{attribute 'reflection'} 
FUNCTION_BLOCK FB_Component IMPLEMENTS I_Component
VAR_INPUT
	fbInfo:						FB_Info(sInstancePath, eState);
	fbEvent:					FB_Event(THIS^);
END_VAR
VAR_OUTPUT
END_VAR
VAR
    {attribute 'hide'}
	{attribute 'instance-path'} 
    {attribute 'noinit'}
    sInstancePath:				STRING(255);	
	eStateRequest:				E_State;
	eState:						E_State;
    {attribute 'hide'}
	eStatePrevious:				E_State;
END_VAR


// Get Infos
fbInfo();

// Events
fbEvent();

// Handle PackML requests and states
CASE eState OF
	E_State.Undefined:
		IF M_Undefined() THEN
			eState:= E_State.Aborting;					
		END_IF
		
	E_State.Aborting:
		IF M_Aborting() THEN
			eState:= E_State.Aborted;	
		END_IF
		
	E_State.Aborted:
		IF M_Aborted() THEN
			eState:= E_State.Clearing;					
		END_IF
		// Handle request
		CASE eStateRequest OF
			E_State.Clearing, E_State.Stopped, E_State.Idle:
				eState:= E_State.Clearing;					
		END_CASE	

	E_State.Clearing:
		IF M_Clearing() THEN
			eState:= E_State.Stopped;			
		END_IF	

	E_State.Stopped:
		IF M_Stopped() THEN
			eState:= E_State.Resetting;				
		END_IF
		// Handle request
		CASE eStateRequest OF
			E_State.Resetting, E_State.Idle:
				eState:= E_State.Resetting;					
			E_State.Aborted, E_State.Aborting:
				eState:= E_State.Aborting;						
		END_CASE
		
	E_State.Resetting:
		IF M_Resetting() THEN
			eState:= E_State.Idle;
		END_IF
		// Handle request
		CASE eStateRequest OF
			E_State.Stopping, E_State.Stopped:
				eState:= E_State.Stopping;					
			E_State.Aborting, E_State.Aborted:
				eState:= E_State.Aborting;						
		END_CASE	
		
	E_State.Idle:
		M_Idle();
		// Handle request
		CASE eStateRequest OF
			E_State.Starting, E_State.Execute:
				eState:= E_State.Starting;
			E_State.Stopping, E_State.Stopped:
				eState:= E_State.Stopping;					
			E_State.Aborting, E_State.Aborted:
				eState:= E_State.Aborting;						
		END_CASE
		
	E_State.Starting:
		IF M_Starting() THEN
			eState:= E_State.Execute;	
		END_IF
		// Handle request
		CASE eStateRequest OF
			E_State.Stopping, E_State.Stopped:
				eState:= E_State.Stopping;					
			E_State.Aborting, E_State.Aborted:
				eState:= E_State.Aborting;						
		END_CASE			

	E_State.Execute:
		IF M_Execute() THEN
			// Wait for state complete
			CASE eStateRequest OF
				E_State.Completing, E_State.Complete:
					eState:= E_State.Completing;					
			END_CASE	
		END_IF
		// Handle request
		CASE eStateRequest OF
			E_State.Suspending, E_State.Suspend:
				eState:= E_State.Suspending;
			E_State.Holding, E_State.Held:
				eState:= E_State.Holding;
		 	E_State.Completing, E_State.Complete:
				eState:= E_State.Completing;
			E_State.Stopping, E_State.Stopped:
				eState:= E_State.Stopping;					
			E_State.Aborting, E_State.Aborted:
				eState:= E_State.Aborting;						
		END_CASE	

	E_State.Suspend:
		IF M_Suspend() THEN
			eState:= E_State.Unsuspending;			
		END_IF
		// Handle request
		CASE eStateRequest OF
			E_State.Starting, E_State.Execute, E_State.Unsuspending:
				eState:= E_State.Starting;
			E_State.Stopping, E_State.Stopped:
				eState:= E_State.Stopping;					
			E_State.Aborting, E_State.Aborted:
				eState:= E_State.Aborting;						
		END_CASE		

		
	E_State.Stopping:
		IF M_Stopping() THEN
			eState:= E_State.Stopped;	
		END_IF
		// Handle request
		CASE eStateRequest OF	
			E_State.Aborting, E_State.Aborted:
				eState:= E_State.Aborting;						
		END_CASE			
	
	E_State.Holding:
		IF M_Holding() THEN
			eState:= E_State.Held;	
		END_IF
		// Handle request
		CASE eStateRequest OF
			E_State.Stopping, E_State.Stopped:
				eState:= E_State.Stopping;					
			E_State.Aborting, E_State.Aborted:
				eState:= E_State.Aborting;						
		END_CASE		
		
	E_State.Held:
		IF M_Held() THEN
			eState:= E_State.Unholding;			
		END_IF
		// Handle request
		CASE eStateRequest OF
			E_State.Stopping, E_State.Stopped:
				eState:= E_State.Stopping;					
			E_State.Aborting, E_State.Aborted:
				eState:= E_State.Aborting;						
		END_CASE		
		
	E_State.Unholding:
		IF M_Unholding() THEN
			eState:= E_State.Execute;
		END_IF
		// Handle request
		CASE eStateRequest OF
			E_State.Stopping, E_State.Stopped:
				eState:= E_State.Stopping;					
			E_State.Aborting, E_State.Aborted:
				eState:= E_State.Aborting;						
		END_CASE
		
	E_State.Suspending:
		IF M_Suspending() THEN
			eState:= E_State.Suspend;
		END_IF
		// Handle request
		CASE eStateRequest OF
			E_State.Stopping, E_State.Stopped:
				eState:= E_State.Stopping;					
			E_State.Aborting, E_State.Aborted:
				eState:= E_State.Aborting;						
		END_CASE	
		
	E_State.Unsuspending:
		IF M_Unsuspending() THEN
			eState:= E_State.Execute;
		END_IF
		// Handle request
		CASE eStateRequest OF
			E_State.Stopping, E_State.Stopped:
				eState:= E_State.Stopping;					
			E_State.Aborting, E_State.Aborted:
				eState:= E_State.Aborting;						
		END_CASE	
		
	E_State.Completing:
		IF M_Completing() THEN
			eState:= E_State.Complete;
		END_IF
		// Handle request
		CASE eStateRequest OF
			E_State.Stopping, E_State.Stopped:
				eState:= E_State.Stopping;					
			E_State.Aborting, E_State.Aborted:
				eState:= E_State.Aborting;						
		END_CASE
		
	E_State.Complete:
		IF M_Complete() THEN
			eState:= E_State.Resetting;		
		END_IF
		// Handle request
		CASE eStateRequest OF
			E_State.Resetting, E_State.Idle:
				eState:= E_State.Stopping;		
			E_State.Stopping, E_State.Stopped:
				eState:= E_State.Stopping;					
			E_State.Aborting, E_State.Aborted:
				eState:= E_State.Aborting;						
		END_CASE
	
END_CASE
CASE eStateRequest OF
	E_State.Resetting:
		M_Reset();
END_CASE

CASE eState OF
	E_State.Idle, E_State.Complete, E_State.Held, E_State.Suspend, E_State.Aborted, E_State.Stopped:
		M_Reset();
END_CASE

// Detect state changed
IF eStatePrevious <> eState THEN
	M_StateChanged();
	eStateRequest:= eState;
	eStatePrevious:= eState;	
END_IF

METHOD PROTECTED M_Aborted : BOOL
VAR_INPUT
END_VAR
// State Aborted
M_Aborted:= True;
END_METHOD

METHOD PROTECTED M_Aborting : BOOL
VAR_INPUT
END_VAR
// State Aborting
M_Aborting:= True;
END_METHOD

METHOD PROTECTED M_Clearing : BOOL
VAR_INPUT
END_VAR
// State Clearing
M_Clearing:= True;
END_METHOD

METHOD PROTECTED M_Complete : BOOL
VAR_INPUT
END_VAR
// State Complete
M_Complete:= TRUE;
END_METHOD

METHOD PROTECTED M_Completing : BOOL
VAR_INPUT
END_VAR
// State Completing
M_Completing:= True;
END_METHOD

METHOD PROTECTED M_Execute : BOOL
VAR_INPUT
END_VAR
// State Execute
END_METHOD

METHOD PROTECTED M_Held : BOOL
VAR_INPUT
END_VAR
// State Held
M_Held:= TRUE;
END_METHOD

METHOD PROTECTED M_Holding : BOOL
VAR_INPUT
END_VAR
// State Holding
M_Holding:= True;
END_METHOD

METHOD PROTECTED M_Idle : BOOL
VAR_INPUT
END_VAR
// State Idle
END_METHOD

METHOD PUBLIC M_Request : BOOL
VAR_INPUT
	eRequest:	E_Request;
END_VAR
CASE eRequest OF
	E_Request.Undefined:
		M_Request:= FALSE;
		
	E_Request.Complete:
		eStateRequest:= E_State.Completing;
		M_Request:= eState = E_State.Complete;
		
	E_Request.Clear:
		eStateRequest:= E_State.Clearing;
		M_Request:= eState = E_State.Stopped;
		
	E_Request.Reset:
		eStateRequest:= E_State.Resetting;
		M_Request:= eState = E_State.Idle;
	
	E_Request.Start, E_Request.Unhold, E_Request.Unsuspend:
		eStateRequest:= E_State.Execute;
		M_Request:= eState = E_State.Execute;
		
	E_Request.Stop:
		eStateRequest:= E_State.Stopping;	
		M_Request:= eState = E_State.Stopped;
		
	E_Request.Hold:;
		eStateRequest:= E_State.Held;	
		M_Request:= eState = E_State.Held;
		
	E_Request.Suspend:;
		eStateRequest:= E_State.Suspend;	
		M_Request:= eState = E_State.Suspend;
		
	E_Request.Abort:
		eStateRequest:= E_State.Aborted;	
		M_Request:= eState = E_State.Aborted;
		
END_CASE
END_METHOD

METHOD PROTECTED M_Reset : BOOL
VAR_INPUT
END_VAR
END_METHOD

METHOD PROTECTED M_Resetting : BOOL
VAR_INPUT
END_VAR
// State Resetting
M_Resetting:= True;
END_METHOD

METHOD PROTECTED M_Starting : BOOL
VAR_INPUT
END_VAR
// State Starting
M_Starting:= True;
END_METHOD

METHOD PROTECTED M_StateChanged : BOOL
VAR_INPUT
END_VAR
END_METHOD

METHOD PROTECTED M_Stopped : BOOL
VAR_INPUT
END_VAR
// State Clearing
END_METHOD

METHOD PROTECTED M_Stopping : BOOL
VAR_INPUT
END_VAR
// State Stopping
M_Stopping:= True;
END_METHOD

METHOD PROTECTED M_Suspend : BOOL
VAR_INPUT
END_VAR
// State Suspend
M_Suspend:= TRUE;
END_METHOD

METHOD PROTECTED M_Suspending : BOOL
VAR_INPUT
END_VAR
// State Suspending
M_Suspending:= True;
END_METHOD

METHOD PROTECTED M_Undefined : BOOL;
VAR_INPUT
END_VAR
// State Undefined
M_Undefined:= True;
END_METHOD

METHOD PROTECTED M_Unholding : BOOL
VAR_INPUT
END_VAR
// State Unholding
M_Unholding:= True;
END_METHOD

METHOD PROTECTED M_Unsuspending : BOOL
VAR_INPUT
END_VAR
// State Unsuspending
M_Unsuspending:= True;
END_METHOD

PROPERTY PUBLIC P_Event : I_Event
GET
P_Event:= fbEvent;
END_GET
END_PROPERTY

PROPERTY PUBLIC P_Info : I_Info
GET
P_Info:= fbInfo;
END_GET
END_PROPERTY

END_FUNCTION_BLOCK

(* stored: Version 1.1.0.1
   POU FB_Component: Id {4a8fdfc8-695a-4bb4-a889-b0289c0a194c}, SpecialFunc None
   Folder States: Id {bb7123de-6478-4234-9ee4-651df2b9bc25}
   Method M_Aborted: Id {851e7e88-c79a-42ec-971c-1651bbdcd922}
   Method M_Aborting: Id {2544540d-284d-4bb6-9092-9fb2d57b609d}
   Method M_Clearing: Id {7ca46105-e5ff-4ca0-9f27-b897928eeabb}
   Method M_Complete: Id {36dec38b-240d-4516-a167-d73475e82b56}
   Method M_Completing: Id {d7947499-dc81-4824-8eb2-1f31346a18c9}
   Method M_Execute: Id {7b4271f8-8ab7-4ecd-8059-762441f55350}
   Method M_Held: Id {897a0d48-e739-4f14-8313-6cf76e869ecc}
   Method M_Holding: Id {7537786e-be59-43f8-af14-91fbd68626c4}
   Method M_Idle: Id {9f0f7190-6eb5-4f18-a951-5893e9af72d3}
   Method M_Request: Id {ccb3d941-e869-469e-bebe-469135ac244b}
   Method M_Reset: Id {086635ef-5800-4505-9adb-437f3dabe309}
   Method M_Resetting: Id {ef3b38ac-7092-48f4-bd93-3280fba28638}
   Method M_Starting: Id {0a285b28-e7e5-4050-bddf-636ff865dc31}
   Method M_StateChanged: Id {fed7d462-efbd-4bae-956c-60dd99530457}
   Method M_Stopped: Id {3035f166-5ee3-4891-8715-c804b18a321e}
   Method M_Stopping: Id {044bf6dd-28e6-4ae0-8f4c-d70b321a375a}
   Method M_Suspend: Id {a3699799-24ae-4f9f-afe8-4644b106fc28}
   Method M_Suspending: Id {d734c7b7-046c-4574-8d27-bb51a30e04e7}
   Method M_Undefined: Id {54f2b561-b89f-47f6-a504-ad1a94f7dafa}
   Method M_Unholding: Id {169fe3b1-c782-410c-a757-900a6ea2c822}
   Method M_Unsuspending: Id {a44bfedf-60a0-4908-9b14-58843306f08b}
   Property P_Event: Id {3b935d9d-6278-4dc9-a359-4ee7f1c69123}
   Get Get: Id {29792270-b47c-4141-a645-41c0781f774b}
   Property P_Info: Id {6e421f29-8ecf-4944-bc3a-6ca6205a23ab}
   Get Get: Id {f1bd3bb2-b46e-4fac-8458-ce900be7323b} *)
